PROGRAM prg_VerschalenDisplay
VAR
	nPotentioMeter		AT		%I*		:INT;
	
	nPotPower			AT		%Q*		:INT := 32767; //Potentiometer voeden met 5V
	nWaarde				AT		%Q*		:INT;
END_VAR

nWaarde := nPotentioMeter * 1000 / 32767;

//Misschien zelfs beter maar onnodig moeilijke oplossing:
//	nWaarde := REAL_TO_INT(INT_TO_REAL(nPotentioMeter) * 1000 / 32767);

END_PROGRAM

(* stored: Version 1.1.0.1, ProductVersion 3.1.4024.15
   POU prg_VerschalenDisplay: Id {1f1518e3-7892-4b3f-92b4-c0836a4d9eb1}, SpecialFunc None *)
